(* PLC project OOP_Curso, Beckhoff Automation GmbH TwinCAT PLC Control 3.5.13.21 *)
(* stored: creationDateTime 2023-06-17T13:41:32.760416, modificationDateTime 2023-06-17T13:41:32.7672534 *)

INTERFACE I_Delayable EXTENDS __SYSTEM.IQueryInterface
PROPERTY tOffDelay : TIME
END_PROPERTY
PROPERTY tOnDelay : TIME
END_PROPERTY
END_INTERFACE

INTERFACE I_Dimmable EXTENDS __SYSTEM.IQueryInterface
METHOD M_RecallMinLevel
VAR_INPUT
END_VAR
END_METHOD
METHOD M_SetControlLevel
VAR_INPUT
	nControlLevel	:	BYTE;
END_VAR
END_METHOD
PROPERTY nControlLevel : BYTE
END_PROPERTY
PROPERTY nMaxLevel : BYTE
END_PROPERTY
PROPERTY nMinLevel : BYTE
END_PROPERTY
END_INTERFACE

INTERFACE I_Light EXTENDS __SYSTEM.IQueryInterface
METHOD M_Off
VAR_INPUT
END_VAR
END_METHOD
METHOD M_On
VAR_INPUT
END_VAR
END_METHOD
PROPERTY bControlLevel : BOOL
END_PROPERTY
END_INTERFACE

FUNCTION_BLOCK PUBLIC FB_DelayedLight EXTENDS FB_Light IMPLEMENTS I_Delayable
VAR_INPUT
END_VAR
VAR_OUTPUT
END_VAR
VAR
	_tOnDelay			:	TIME;
	_tOffDelay			:	TIME;
	tonOnDelay			:	TON;
	tonOffDelay			:	TON;
	bStartOnDelay		:	BOOL;
	bStartOffDelay		:	BOOL;
	nStep				:	INT;
END_VAR

            rtrigOn(CLK := bOn);
IF (rtrigOn.Q) THEN
	M_On();
END_IF

rtrigOff(CLK := bOff);
IF (rtrigOff.Q) THEN
	M_Off();
END_IF

CASE nStep OF
	0:
		IF ((bStartOnDelay AND nStep = 0)) THEN
			tonOnDelay(IN := FALSE);
			nStep := 10;
		END_IF
		IF ((bStartOffDelay AND nStep = 0)) THEN
			tonOffDelay(IN := FALSE);
			nStep := 20;
		END_IF
	10:
		tonOnDelay(IN := TRUE, pt := tOnDelay);
		IF (tonOnDelay.Q) THEN
			SUPER^._bControlLevel := TRUE;
			bStartOnDelay := FALSE;
			nStep := 0;
		END_IF
	20:
		tonOffDelay(IN := TRUE, pt := tOffDelay);
		IF (tonOffDelay.Q) THEN
			SUPER^._bControlLevel := FALSE;
			bStartOffDelay := FALSE;
			nStep := 0;
		END_IF
END_CASE

bControl := bControlLevel;

          

METHOD PUBLIC FB_init : BOOL
VAR_INPUT
	bInitRetains : BOOL; // if TRUE, the retain variables are initialized (warm start / cold start)
	bInCopyCode : BOOL;  // if TRUE, the instance afterwards gets moved into the copy code (online change)
END_VAR
                  _tOnDelay := T#1S;
_tOffDelay := T#2S;

                
END_METHOD

METHOD PUBLIC M_Off
                  bStartOffDelay := TRUE;
                
END_METHOD

METHOD PUBLIC M_On
                  bStartOnDelay := TRUE;
                
END_METHOD

PROPERTY tOffDelay : TIME
GET
VAR
END_VAR
                    tOffDelay := _tOffDelay;
                  
END_GET
SET
VAR
END_VAR
                    _tOffDelay := tOffDelay;
                  
END_SET
END_PROPERTY

PROPERTY tOnDelay : TIME
GET
VAR
END_VAR
                    tOnDelay := _tOnDelay;
                  
END_GET
SET
VAR
END_VAR
                    _tOnDelay := tOnDelay;
                  
END_SET
END_PROPERTY
END_FUNCTION_BLOCK

FUNCTION_BLOCK PUBLIC FB_DimmingLight EXTENDS FB_Light IMPLEMENTS I_Dimmable
VAR_INPUT
	bRecallMinLevel			:	BOOL;
	bSetControlLevel		:	BOOL;
	nSetControlLevel		:	BYTE;
END_VAR
VAR_OUTPUT
	nControl				:	BYTE;
END_VAR
VAR
	rtrigRecallMinLevel		:	R_TRIG;
	rtrigSetControlLevel	:	R_TRIG;
	_nControlLevel			:	BYTE;
	_nMinLevel				:	BYTE;
	_nMaxLevel				:	BYTE;
END_VAR

            rtrigOn(CLK := bOn);
IF (rtrigOn.Q) THEN
	M_On();
END_IF

rtrigOff(CLK := bOff);
IF (rtrigOff.Q) THEN
	M_Off();
END_IF

rtrigRecallMinLevel(CLK := bRecallMinLevel);
IF (rtrigRecallMinLevel.Q) THEN
	M_RecallMinLevel();
END_IF

rtrigSetControlLevel(CLK := bSetControlLevel);
IF (rtrigSetControlLevel.Q) THEN
	M_SetControlLevel(nSetControlLevel);
END_IF

bControl := bControlLevel;
nControl := nControlLevel;


          

METHOD PUBLIC FB_init : BOOL
VAR_INPUT
	bInitRetains : BOOL; // bei TRUE werden die Retain-Variablen initialisiert (Warmstart / Kaltstart)
	bInCopyCode : BOOL;  // bei TRUE wird die Instanz anschließend in den Copy-Code kopiert (Online Change)
END_VAR
                  _nMinLevel := 10;
_nMaxLevel := 100;

                
END_METHOD

METHOD PUBLIC M_Off
                  _bControlLevel := FALSE;
_nControlLevel := 0;
                
END_METHOD

METHOD PUBLIC M_On
                  _bControlLevel := TRUE;
_nControlLevel := _nMaxLevel;
                
END_METHOD

METHOD PUBLIC M_RecallMinLevel
                  _bControlLevel := TRUE;
_nControlLevel := _nMinLevel;
                
END_METHOD

METHOD PUBLIC M_SetControlLevel
VAR_INPUT
	nControlLevel	: BYTE;
END_VAR
                  IF (nControlLevel = 0) THEN
	THIS^.M_Off();
ELSIF ((nControlLevel > 0) AND (nControlLevel <= _nMinLevel)) THEN
	_bControlLevel := TRUE;
	_nControlLevel := _nMinLevel;	
ELSIF ((nControlLevel > _nMinLevel) AND (nControlLevel <= _nMaxLevel)) THEN
	_bControlLevel := TRUE;
	_nControlLevel := nControlLevel;	
ELSE
	_bControlLevel := TRUE;
	_nControlLevel := _nMaxLevel;	
END_IF

                
END_METHOD

PROPERTY nControlLevel : BYTE
GET
VAR
END_VAR
                    nControlLevel := _nControlLevel;
                  
END_GET
SET
VAR
END_VAR
                    
                  
END_SET
END_PROPERTY

PROPERTY nMaxLevel : BYTE
GET
VAR
END_VAR
                    nMaxLevel := _nMaxLevel;
                  
END_GET
SET
VAR
END_VAR
                    _nMaxLevel := nMaxLevel;
                  
END_SET
END_PROPERTY

PROPERTY nMinLevel : BYTE
GET
VAR
END_VAR
                    nMinLevel := _nMinLevel;
                  
END_GET
SET
VAR
END_VAR
                    _nMinLevel := nMinLevel;
                  
END_SET
END_PROPERTY
END_FUNCTION_BLOCK

FUNCTION_BLOCK PUBLIC FB_Light IMPLEMENTS I_Light
VAR_INPUT
	bOn					:	BOOL;
	bOff				:	BOOL;
END_VAR
VAR_OUTPUT
	bControl			:	BOOL;
END_VAR
VAR
	rtrigOn				:	R_TRIG;
	rtrigOff			:	R_TRIG;
	_bControlLevel		:	BOOL;
END_VAR

            rtrigOn(CLK := bOn);
IF (rtrigOn.Q) THEN
	M_On();
END_IF

rtrigOff(CLK := bOff);
IF (rtrigOff.Q) THEN
	M_Off();
END_IF

bControl := bControlLevel;

          

METHOD PUBLIC M_Off
                  _bControlLevel := FALSE;
                
END_METHOD

METHOD PUBLIC M_On
                  _bControlLevel := TRUE;
                
END_METHOD

PROPERTY bControlLevel : BOOL
GET
VAR
END_VAR
                    bControlLevel := _bControlLevel;
                  
END_GET
SET
VAR
END_VAR
                    
                  
END_SET
END_PROPERTY
END_FUNCTION_BLOCK

FUNCTION_BLOCK PUBLIC FB_RoomController
VAR_INPUT
	bAllOn					:	BOOL;
	bAllOff					:	BOOL;
	bAllCallMinLevel		:	BOOL;
	refLight01				:	REFERENCE TO FB_Light;
	refLight02				:	REFERENCE TO FB_Light;
	refLight03				:	REFERENCE TO FB_Light;
END_VAR
VAR_OUTPUT
	aControlLevel			:	ARRAY [1..3] OF BOOL;
	aDimmLevel				:	ARRAY [1..3] OF BYTE;
END_VAR
VAR
	aILight					:	ARRAY [1..3] OF I_Light;
	aIDimmableLights		:	ARRAY [1..3] OF I_Dimmable;
	rtrigAllOn				:	R_TRIG;
	rtrigAllOff				:	R_TRIG;
	rtrigAllCallMinLevel	:	R_TRIG;
END_VAR

            rtrigAllOn(CLK := bAllOn);
IF (rtrigAllOn.Q) THEN
	AllOn();
END_IF

rtrigAllOff(CLK := bAllOff);
IF (rtrigAllOff.Q) THEN
	AllOff();
END_IF

rtrigAllCallMinLevel(CLK := bAllCallMinLevel);
IF (rtrigAllCallMinLevel.Q) THEN
	AllCallMinLevel();
END_IF

Invoke();

          

ACTION AllCallMinLevel:
                IF (__ISVALIDREF(refLight01)) THEN
	aILight[1] := refLight01;
	IF (__QUERYINTERFACE(aILight[1], aIDimmableLights[1])) THEN
		aIDimmableLights[1].M_RecallMinLevel();
	END_IF
END_IF

IF (__ISVALIDREF(refLight02)) THEN
	aILight[2] := refLight02;
	IF (__QUERYINTERFACE(aILight[2], aIDimmableLights[2])) THEN
		aIDimmableLights[2].M_RecallMinLevel();
	END_IF
END_IF

IF (__ISVALIDREF(refLight03)) THEN
	aILight[3] := refLight03;
	IF (__QUERYINTERFACE(aILight[3], aIDimmableLights[3])) THEN
		aIDimmableLights[3].M_RecallMinLevel();
	END_IF
END_IF
              
END_ACTION

ACTION AllOff:
                IF (__ISVALIDREF(refLight01)) THEN
	refLight01.M_Off();
END_IF
IF (__ISVALIDREF(refLight02)) THEN
	refLight02.M_Off();
END_IF
IF (__ISVALIDREF(refLight03)) THEN
	refLight03.M_Off();
END_IF
              
END_ACTION

ACTION AllOn:
                IF (__ISVALIDREF(refLight01)) THEN
	refLight01.M_On();
END_IF
IF (__ISVALIDREF(refLight02)) THEN
	refLight02.M_On();
END_IF
IF (__ISVALIDREF(refLight03)) THEN
	refLight03.M_On();
END_IF
              
END_ACTION

ACTION Invoke:
                IF (__ISVALIDREF(refLight01)) THEN
	refLight01();
	aControlLevel[1] := refLight01.bControlLevel;	
	aILight[1] := refLight01;
	IF (__QUERYINTERFACE(aILight[1], aIDimmableLights[1])) THEN
		aDimmLevel[1] := aIDimmableLights[1].nControlLevel;
	END_IF
END_IF
IF (__ISVALIDREF(refLight02)) THEN
	refLight02();
	aControlLevel[2] := refLight02.bControlLevel;
	aILight[2] := refLight02;
	IF (__QUERYINTERFACE(aILight[2], aIDimmableLights[2])) THEN
		aDimmLevel[2] := aIDimmableLights[2].nControlLevel;
	END_IF
END_IF
IF (__ISVALIDREF(refLight03)) THEN
	refLight03();
	aControlLevel[3] := refLight03.bControlLevel;
	aILight[3] := refLight03;
	IF (__QUERYINTERFACE(aILight[3], aIDimmableLights[3])) THEN
		aDimmLevel[3] := aIDimmableLights[3].nControlLevel;
	END_IF
END_IF

              
END_ACTION
END_FUNCTION_BLOCK

FUNCTION_BLOCK FB_MyLight EXTENDS FB_Light IMPLEMENTS I_Delayable, I_Dimmable
VAR_INPUT
	bRecallMinLevel			:	BOOL;
	bSetControlLevel		:	BOOL;
	nSetControlLevel		:	BYTE;
END_VAR
VAR_OUTPUT
	nControl				:	BYTE;
END_VAR
VAR
	rtrigRecallMinLevel		:	R_TRIG;
	rtrigSetControlLevel	:	R_TRIG;
	fbDimmingLight			:	FB_DimmingLight;
	fbDelayedLight			:	FB_DelayedLight;
	_nControlLevel			:	BYTE;
END_VAR

            rtrigOn(CLK := bOn);
IF (rtrigOn.Q) THEN
	M_On();
END_IF

rtrigOff(CLK := bOff);
IF (rtrigOff.Q) THEN
	M_Off();
END_IF

rtrigRecallMinLevel(CLK := bRecallMinLevel);
IF (rtrigRecallMinLevel.Q) THEN
	M_RecallMinLevel();
END_IF

rtrigSetControlLevel(CLK := bSetControlLevel);
IF (rtrigSetControlLevel.Q) THEN
	M_SetControlLevel(nSetControlLevel);
END_IF

fbDimmingLight();
fbDelayedLight();
_bControlLevel := fbDelayedLight.bControlLevel;
IF (_bControlLevel) THEN
	_nControlLevel := fbDimmingLight.nControlLevel;
ELSE
	_nControlLevel := 0;		
END_IF

bControl := bControlLevel;
nControl := nControlLevel;


          

METHOD M_Off
                  fbDimmingLight.M_Off();
fbDelayedLight.M_Off();

                
END_METHOD

METHOD M_On
                  fbDimmingLight.M_On();
fbDelayedLight.M_On();

                
END_METHOD

METHOD M_RecallMinLevel
                  fbDimmingLight.M_RecallMinLevel();
fbDelayedLight.M_On();

                
END_METHOD

METHOD M_SetControlLevel
VAR_INPUT
	nControlLevel: BYTE;
END_VAR
                  fbDimmingLight.M_SetControlLevel(nControlLevel);
IF (nControlLevel = 0) THEN
	fbDelayedLight.M_Off();
ELSE
	fbDelayedLight.M_On();
END_IF

                
END_METHOD

PROPERTY bControlLevel : BOOL
GET
                    bControlLevel := _bControlLevel;
                  
END_GET
SET
                    
                  
END_SET
END_PROPERTY

PROPERTY nControlLevel : BYTE
GET
                    nControlLevel := _nControlLevel;
                  
END_GET
SET
                    
                  
END_SET
END_PROPERTY

PROPERTY nMaxLevel : BYTE
GET
                    nMaxLevel := THIS^.fbDimmingLight.nMaxLevel;
                  
END_GET
SET
                    THIS^.fbDimmingLight.nMaxLevel := nMaxLevel;
                  
END_SET
END_PROPERTY

PROPERTY nMinLevel : BYTE
GET
                    nMinLevel := THIS^.fbDimmingLight.nMinLevel;
                  
END_GET
SET
                    THIS^.fbDimmingLight.nMaxLevel := nMaxLevel;
                  
END_SET
END_PROPERTY

PROPERTY tOffDelay : TIME
GET
                    
                  
END_GET
SET
                    
                  
END_SET
END_PROPERTY

PROPERTY tOnDelay : TIME
GET
                    
                  
END_GET
SET
                    
                  
END_SET
END_PROPERTY
END_FUNCTION_BLOCK

PROGRAM P_DelayedLight_Test_CFC
VAR
	fbDelayedLight		:	FB_DelayedLight;
	bOn					:	BOOL;
	bOff				:	BOOL;
	bControlLevel		:	BOOL;
END_VAR

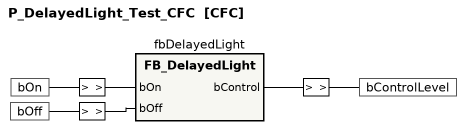
(* CFC diagram, written out as Structured Text *)
fbDelayedLight(bOn := bOn, bOff := bOff);
bControlLevel := fbDelayedLight.bControl;
END_PROGRAM

PROGRAM P_DelayedLight_Test_ST
VAR
	fbDelayedLight		:	FB_DelayedLight;
	bOn					:	BOOL;
	bOff				:	BOOL;
	bControlLevel		:	BOOL;	
END_VAR

            fbDelayedLight();

IF (bOn) THEN
	fbDelayedLight.M_On();
	bOn := FALSE;
END_IF
IF (bOff) THEN
	fbDelayedLight.M_Off();
	bOff := FALSE;
END_IF

bControlLevel := fbDelayedLight.bControlLevel;


          
END_PROGRAM

PROGRAM P_DimmingLight_Test_CFC
VAR
	fbDimmingLight		:	FB_DimmingLight;
	bOn					:	BOOL;
	bOff				:	BOOL;
	bRecallMinLevel		:	BOOL;
	bSetControlLevel	:	BOOL;
	nSetControlLevel	:	BYTE;
	bControlLevel		:	BOOL;
	nControlLevel		:	BYTE;
END_VAR

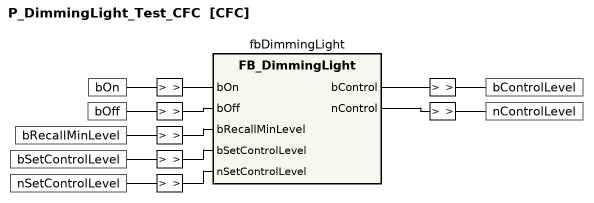
(* CFC diagram, written out as Structured Text *)
fbDimmingLight(bOn := bOn, bOff := bOff, bRecallMinLevel := bRecallMinLevel, bSetControlLevel := bSetControlLevel, nSetControlLevel := nSetControlLevel);
bControlLevel := fbDimmingLight.bControl;
nControlLevel := fbDimmingLight.nControl;
END_PROGRAM

PROGRAM P_DimmingLight_Test_ST
VAR
	fbDimmingLight		:	FB_DimmingLight;
	bOn					:	BOOL;
	bOff				:	BOOL;
	bRecallMinLevel		:	BOOL;
	bSetControlLevel	:	BOOL;
	nSetControlLevel	:	BYTE;
	bControlLevel		:	BOOL;
	nControlLevel		:	BYTE;
END_VAR

            fbDimmingLight();

IF (bOn) THEN
	fbDimmingLight.M_On();
	bOn := FALSE;
END_IF
IF (bOff) THEN
	fbDimmingLight.M_Off();
	bOff := FALSE;
END_IF
IF (bRecallMinLevel) THEN
	fbDimmingLight.M_RecallMinLevel();
	bRecallMinLevel := FALSE;
END_IF
IF (bSetControlLevel) THEN
	fbDimmingLight.M_SetControlLevel(nSetControlLevel);
	bSetControlLevel := FALSE;
END_IF

bControlLevel := fbDimmingLight.bControlLevel;
nControlLevel := fbDimmingLight.nControlLevel;



          
END_PROGRAM

PROGRAM P_Light_Test_CFC
VAR
	fbLight				:	FB_Light;
	bOn					:	BOOL;
	bOff				:	BOOL;
	bControlLevel		:	BOOL;
END_VAR

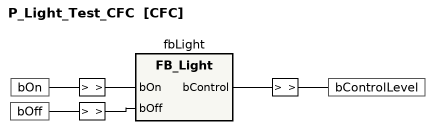
(* CFC diagram, written out as Structured Text *)
fbLight(bOn := bOn, bOff := bOff);
bControlLevel := fbLight.bControl;
END_PROGRAM

PROGRAM P_Light_Test_ST
VAR
	fbLight				:	FB_Light;
	bOn					:	BOOL;
	bOff				:	BOOL;
	bControlLevel		:	BOOL;	
END_VAR

            fbLight();

IF (bOn) THEN
	fbLight.M_On();
	bOn := FALSE;
END_IF
IF (bOff) THEN
	fbLight.M_Off();
	bOff := FALSE;
END_IF

bControlLevel := fbLight.bControlLevel;


          
END_PROGRAM

PROGRAM P_MyLight_Test_CFC
VAR
	fbMyLight			:	FB_MyLight1;
	bOn					:	BOOL;
	bOff				:	BOOL;
	bRecallMinLevel		:	BOOL;
	bSetControlLevel	:	BOOL;
	nSetControlLevel	:	BYTE;
	bControlLevel		:	BOOL;
	nControlLevel		:	BYTE;
END_VAR

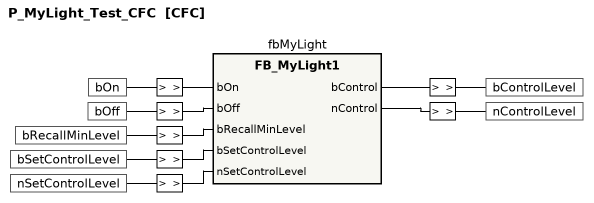
(* CFC diagram, written out as Structured Text *)
bControlLevel := fbMyLight.bControl;
nControlLevel := fbMyLight.nControl;
fbMyLight(bOn := bOn, bOff := bOff, bRecallMinLevel := bRecallMinLevel, bSetControlLevel := bSetControlLevel, nSetControlLevel := nSetControlLevel);
END_PROGRAM

PROGRAM P_MyLight_Test_ST
VAR
	fbMyLight			:	FB_MyLight1;
	bOn					:	BOOL;
	bOff				:	BOOL;
	bRecallMinLevel		:	BOOL;
	bSetControlLevel	:	BOOL;
	nSetControlLevel	:	BYTE;
	bControlLevel		:	BOOL;
	nControlLevel		:	BYTE;
END_VAR

            fbMyLight();

IF (bOn) THEN
	fbMyLight.M_On();
	bOn := FALSE;
END_IF
IF (bOff) THEN
	fbMyLight.M_Off();
	bOff := FALSE;
END_IF
IF (bRecallMinLevel) THEN
	fbMyLight.M_RecallMinLevel();
	bRecallMinLevel := FALSE;
END_IF
IF (bSetControlLevel) THEN
	fbMyLight.M_SetControlLevel(nSetControlLevel);
	bSetControlLevel := FALSE;
END_IF

bControlLevel := fbMyLight.bControlLevel;
nControlLevel := fbMyLight.nControlLevel;



          
END_PROGRAM

PROGRAM P_RoomController_Test_CFC
VAR
	fbRoomController	:	FB_RoomController;
	fbmyLight			:	FB_MyLight1;
	fbDelayedLight		:	FB_DelayedLight;
	fbDimmingLight		:	FB_DimmingLight;
	bAllOn				:	BOOL;
	bAllOff				:	BOOL;
	bAllCallMinLevel	:	BOOL;
	aControlLevel		:	ARRAY [1..3] OF BOOL;
	aDimmLevel			:	ARRAY [1..3] OF BYTE;
END_VAR

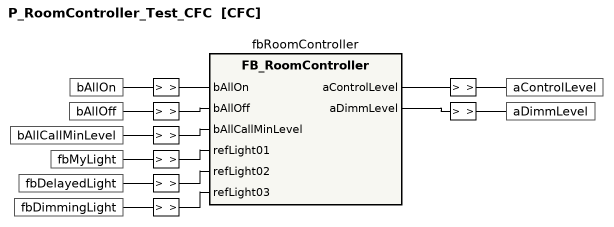
(* CFC diagram, written out as Structured Text *)
fbRoomController(bAllOn := bAllOn, bAllOff := bAllOff, bAllCallMinLevel := bAllCallMinLevel, refLight01 := fbMyLight, refLight02 := fbDelayedLight, refLight03 := fbDimmingLight);
aControlLevel := fbRoomController.aControlLevel;
aDimmLevel := fbRoomController.aDimmLevel;
END_PROGRAM

PROGRAM P_RoomController_Test_ST
VAR
	fbRoomController	:	FB_RoomController;
	fbMyLight			:	FB_MyLight1;
	fbDelayedLight		:	FB_DelayedLight;
	fbDimmingLight		:	FB_DimmingLight;
	bAllOn				:	BOOL;
	bAllOff				:	BOOL;
	bAllCallMinLevel	:	BOOL;
	aControlLevel		:	ARRAY [1..3] OF BOOL;
	aDimmLevel			:	ARRAY [1..3] OF BYTE;
END_VAR

            fbRoomController(bAllOn	:= bAllOn,
				 bAllOff := bAllOff,
				 bAllCallMinLevel := bAllCallMinLevel,
				 refLight01 := fbMyLight,
				 refLight02 := fbDelayedLight,
				 refLight03 := fbDimmingLight,
				 aControlLevel => aControlLevel,
				 aDimmLevel => aDimmLevel);

          
END_PROGRAM

PROGRAM _16_Interface_vs_Herencia
VAR

END_VAR

            P_Light_Test_ST();
P_Light_Test_CFC();

P_DelayedLight_Test_ST();
P_DelayedLight_Test_CFC();

P_DimmingLight_Test_ST();
P_DimmingLight_Test_CFC();

P_MyLight_Test_ST();
P_MyLight_Test_CFC();

P_RoomController_Test_ST();
P_RoomController_Test_CFC();
          
END_PROGRAM

FUNCTION_BLOCK FB_MyLight1 EXTENDS FB_Light IMPLEMENTS I_Delayable, I_Dimmable
VAR_INPUT
	bRecallMinLevel			:	BOOL;
	bSetControlLevel		:	BOOL;
	nSetControlLevel		:	BYTE;
END_VAR
VAR_OUTPUT
	nControl				:	BYTE;
END_VAR
VAR
	rtrigRecallMinLevel		:	R_TRIG;
	rtrigSetControlLevel	:	R_TRIG;
	fbDimmingLight			:	FB_DimmingLight;
	fbDelayedLight			:	FB_DelayedLight;
	_nControlLevel			:	BYTE;
END_VAR

            rtrigOn(CLK := bOn);
IF (rtrigOn.Q) THEN
	M_On();
END_IF

rtrigOff(CLK := bOff);
IF (rtrigOff.Q) THEN
	M_Off();
END_IF

rtrigRecallMinLevel(CLK := bRecallMinLevel);
IF (rtrigRecallMinLevel.Q) THEN
	M_RecallMinLevel();
END_IF

rtrigSetControlLevel(CLK := bSetControlLevel);
IF (rtrigSetControlLevel.Q) THEN
	M_SetControlLevel(nSetControlLevel);
END_IF

fbDimmingLight();
fbDelayedLight();
_bControlLevel := fbDelayedLight.bControlLevel;
IF (_bControlLevel) THEN
	_nControlLevel := fbDimmingLight.nControlLevel;
ELSE
	_nControlLevel := 0;		
END_IF

bControl := bControlLevel;
nControl := nControlLevel;


          

METHOD M_Off
                  fbDimmingLight.M_Off();
fbDelayedLight.M_Off();

                
END_METHOD

METHOD M_On
                  fbDimmingLight.M_On();
fbDelayedLight.M_On();

                
END_METHOD

METHOD M_RecallMinLevel
                  fbDimmingLight.M_RecallMinLevel();
fbDelayedLight.M_On();

                
END_METHOD

METHOD M_SetControlLevel
VAR_INPUT
	nControlLevel: BYTE;
END_VAR
                  fbDimmingLight.M_SetControlLevel(nControlLevel);
IF (nControlLevel = 0) THEN
	fbDelayedLight.M_Off();
ELSE
	fbDelayedLight.M_On();
END_IF

                
END_METHOD

PROPERTY bControlLevel : BOOL
GET
                    bControlLevel := _bControlLevel;
                  
END_GET
SET
                    
                  
END_SET
END_PROPERTY

PROPERTY nControlLevel : BYTE
GET
                    nControlLevel := _nControlLevel;
                  
END_GET
SET
                    
                  
END_SET
END_PROPERTY

PROPERTY nMaxLevel : BYTE
GET
                    nMaxLevel := THIS^.fbDimmingLight.nMaxLevel;
                  
END_GET
SET
                    THIS^.fbDimmingLight.nMaxLevel := nMaxLevel;
                  
END_SET
END_PROPERTY

PROPERTY nMinLevel : BYTE
GET
                    nMinLevel := THIS^.fbDimmingLight.nMinLevel;
                  
END_GET
SET
                    THIS^.fbDimmingLight.nMaxLevel := nMaxLevel;
                  
END_SET
END_PROPERTY

PROPERTY tOffDelay : TIME
GET
                    
                  
END_GET
SET
                    
                  
END_SET
END_PROPERTY

PROPERTY tOnDelay : TIME
GET
                    
                  
END_GET
SET
                    
                  
END_SET
END_PROPERTY
END_FUNCTION_BLOCK
